Staubli VAL3: stop.pgx

program stop()
begin
  stopMove()
  resetMotion()
  clearBuffer(sSockPC)
end
